{attribute 'qualified_only'}
VAR_GLOBAL
db1 : BOOL;
Z2 : BOOL;
Db3 : BOOL;
Db4 : BOOL;
Db5 : BOOL;
Db6 : BOOL;
END_VAR

(* stored: Version 1.1.0.1, ProductVersion 3.1.4024.12
   GVL ZONE: Id {3cfa742b-91cd-4ba2-a920-9d694d75432c} *)
